DATA_BLOCK "数据块_1"
{ S7_Optimized_Access := 'FALSE' }
VERSION : 0.1
   STRUCT
      a : Bool;
   END_STRUCT;


BEGIN

END_DATA_BLOCK

